FUNCTION_BLOCK DIV_UINT (* IEC 61131-3 UINT Division *)
  (* Standard: 61131-3 *)
  (* Version 0.0, 2004-12-15, JHC, Rockwell Automation, Converted from SRC format. *)
  (* Compiler header: package fb.rt.plc.math; *)
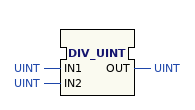
  VAR_INPUT
    IN1 : UINT; (* Dividend *)
    IN2 : UINT; (* Divisor *)
  END_VAR
  VAR_OUTPUT
    OUT : UINT; (* Quotient *)
  END_VAR
END_FUNCTION_BLOCK
